(* IEC 61131-3 sources: Dev/Dev_V200/200 (part 15) *)

(* ---- _Nh_Frm_BRW.st ---- *)
FUNCTION _Nh_Frm_Row_BRW {HIDDEN}    : BOOL        // naplni, alebo refreshne objekty jedneho riadka browsu/frame/home
	{ $ IFDEF __NH_WEB }
   VAR_INPUT
      new   : BOOL;
      row   : USINT;
   END_VAR
   VAR_TEMP
		blk	: USINT;
      cp    : USINT;
//      np    : INT;
   END_VAR
   _Nh_Frm_Row_BRW := true;
   IF new THEN
		cp := xR^.h.cf.c;
      IF xL^.obj = 11 AND xR^.h.cf.c = 1 THEN                                           // ZONA domcek       1 ZON -> ROMs
			cp := 3;
		ELSIF xR^.h.new  THEN
			new := false;
      END_IF;
		IF new THEN
      	_Nh_Brw_Row_DSH(row := row, frm := USINT_TO_UINT(aCfg[ cp ].fBr) );   	// nacita FRM a podla DSH pripravi korekcie X,Y
			_Nh_Brw_Row_OBJ(row := row);
	      _Nh_FRM_Read(frm:=246);   	// nacita rozne preddefinovane objekty v riadku	 xR^.o.ob[]
	     	_Nh_Chk_FAV();
   	   CASE xR^.h.cf.c OF
			 0:	;
			50:	// timer - v priebehu refreshu sa nemeni
					xTim	:= xDev;
					memcpyPTR(length:=SIZEOF(NH_OBJ_DAT), source:=ADR(yFrm_246.tim_1), dest:=ADR(xR^.o.ob[6]) );		// nastavi zobrazovanie obrazka typu casovaca nad hlavnou ikonou
					memcpyPTR(length:=SIZEOF(NH_OBJ_DAT), source:=ADR(yFrm_246.e4O1), dest:=ADR(xR^.o.ob[7]) );		// vypne zobrazovanie na stavovou ikonou
			 		x4o   			:= ADR(xR^.o.ob[6]);
					x4o^.obr[2]    :=	yFrm_246.tim_1_typ_obr[ xTim^.cf.typ ];			// podla typu vyberie obrazok
					blk	:= 5;
	      END_CASE;

	   END_IF;
	END_IF;

   CASE xR^.h.cf.c OF

   	0: ;
    	1:	_Nh_Shw_ROM_ROW();
		2: // CAT
		   	_Nh_FRM_Read(frm:=232);
            xR^.o.ob[5].cf.c := 0;
  	         xR^.o.ob[5].cf.n := yFrm_232.cat[xR^.h.cf.n].txt;                                  // cislo textu v 1.riadku
            xR^.o.ob[6].cf.c := 0;
  	         xR^.o.ob[6].cf.n := yFrm_232.cat[xR^.h.cf.n].txt+1;                                  // cislo textu v 2.riadku je za prvym
				IF yFrm_232.cat[xR^.h.cf.n].cmd4 = 0 THEN
					xR^.o.ob[4].wh := 0;
				ELSE
					xR^.o.ob[4].cm := yFrm_232.cat[xR^.h.cf.n].cmd4;
				END_IF
				IF yFrm_232.cat[xR^.h.cf.n].cmd2 = 0 THEN
					xR^.o.ob[2].wh := 0;
				ELSE
					xR^.o.ob[2].cm := yFrm_232.cat[xR^.h.cf.n].cmd2;
				END_IF
				xR^.o.ob[1].cm := yFrm_232.cat[xR^.h.cf.n].cmd1;

            IF xA^.usr= 1 THEN                                                   // pre admina vypise cislo CAT
               xR^.o.ob[7].wh    := 6;
               xR^.o.ob[7].cf.c  := 254;
               xR^.o.ob[7].fmt   := CONCAT(INT_TO_STRINGF(xR^.h.cf.n,'%2u'), '');
            END_IF;
		3:	xR^.o.ob[9].cf.c:=252;										// vypisuje sa nazov domceka (domovskej zony)
				_Nh_Shw_ROM_ROW();
		6: // HET
  				xHet  	:= xDev;
				IF xL^.dsh = 4 THEN
					_Nh_Shw_CPY();
      		ELSE
					_NH_Het_Map_Reg();
//					IF xHet^.io[0].own THEN                // DEV regulovanej teploty
               	IF xRegMod^.wht = 1 THEN
							xR^.o.ob[2].fmt := REAL_TO_STRINGF(xHet^.al.ou.val,'%5.1f°');
						ELSE
							xR^.o.ob[2].fmt := REAL_TO_STRINGF(xHet^.al.ou.val,'%5.0f %%');
						END_IF
//					END_IF ;
					IF xHet^.io[1].own THEN                // ma termoventil
						IF xHet^.io[1].zon THEN             // TVE ma teplotu
							xR^.o.ob[5].fmt := REAL_TO_STRINGF(xHet^.io[1].val,'%5.1f°');
						ELSE
						   xR^.o.ob[5].wh := 0;
						END_IF;
						xHet^.al.lst := true;
					ELSE
		   			xR^.o.ob[5].wh := 0;
						xHet^.al.lst := false;
					END_IF;
//	 			IF xA^.admin = false THEN
	 				IF xM^.set=false OR xA^.UsrRight < 2 THEN
	 					xR^.o.ob[1].cm   := 0;
 						xR^.o.ob[4].fn   := 0;
 						xR^.o.ob[6].fn   := 0;
					END_IF;
				END_IF;
  		47: // HEV
            xHet  := xDev;
				IF xL^.dsh = 4 THEN
					_Nh_Shw_CPY();
         	END_IF;
      		IF xHet^.io[0].own THEN                // aktualne % CO2 zo snimaca
					xR^.o.ob[2].fmt := REAL_TO_STRINGF(xHet^.io[0].val,'%6.0f %%');
				END_IF;
				IF xHet^.io[2].own THEN                // ma termoventil
					xHet^.al.lst := true;
				ELSE
					xHet^.al.lst := false;
				END_IF;
//  	 			IF xA^.admin = false THEN
	 			IF xM^.set=false OR xA^.UsrRight < 2 THEN
 					xR^.o.ob[1].cm   := 0;
	 				xR^.o.ob[4].fn   := 0;											// setup nie je
 					xR^.o.ob[6].fn   := 0;                               	// lst vazby nie su
  				END_IF;
				IF xL^.chk AND xR^.o.ob[4].cf.c > 0 THEN
					IF acfg[xR^.o.ob[4].cf.c].tgrp = 15 THEN
 						xR^.o.ob[7].wh   := 0;                      			// ked je vo vazbe PIR, vypnu sa predvolby a zobrazuju sa prvky PIR
					END_IF;
				END_IF;

		7: // KOT
 			_Nh_Shw_TVE_ROW();

		8: // TVE
 			_Nh_Shw_TVE_ROW();

		9: // CER
 			_Nh_Shw_TVE_ROW();

		15: //PIR
				IF	xR^.h.pir THEN					// je vo vazbe
					;
				ELSIF	_NhxRom(nr := xDev^.cf.rom ,x:=55) THEN
					_Nh_Shw_107_ROM(o:=7, day:=true);
	            _Nh_Frm_STA_OU(obj:=2, o:=8);
					blk	:= 5;
//   				_Nh_DEF_VAR(wh:=20, o:=6, x:=ADR(xDev^.cf.blk) );
				ELSE
					xR^.o.ob[7].wh		:= 0;
				END_IF;

		23: // REK
				 _Nh_Shw_TVE_ROW();

		31: // ROL
				xRol 		:= xDev;
				IF new  THEN                        // pri prvom vstupe do FRM. nacitat iny formular podla menu. n
					xRo		:= ADR(xR^.o.ob[5]);
					IF xR^.h.cf.p=0 THEN
						xR^.h.cf.p := xRol^.cf.par;
					END_IF;
					xRo^.cf	:= xR^.h.cf;
					xRo^.chk	:= xL^.chk;					// priznak vazby
				END_IF;

  	 			IF xM^.set AND xF^.cf.c = 2 AND xF^.cf.n = 3 THEN		// pristupne kopirovanie
		  	 			IF xU^.o[1].fn  = 44 AND xL^.dsh = 1 THEN									// zlte COPY
//      D1_7       : NH_OBJ_4O1 	:= (obj:=1, obr:=[44,38,0,0], cmd:=[0,0,0,0], wxy:=[0,0,0,0],ok:=[0,0,0,0], txt:=[0,0,0,0],  );                          // 5=slider;
//							xR^.o.ob[7]		:= xR^.o.ob[8];
						 	x4o    			:= ADR(xR^.o.ob[8]);
							xR^.o.ob[1].cm 	:= 128;									// click na hlavnu ikonu = oznacovanie
							xR^.o.ob[10].cm 	:= 128;									// nazov
							x4o^.wh			:= 107;
							x4o^.obj			:= 1;
   	 					x4o^.wxy[1]    := 52;
    						x4o^.wxy[2]    := 42;
							x4o^.obr[1]		:= 44;
							x4o^.obr[2]		:= 38;
							x4o^.ok[1] 		:= xU^.o[1].wh = xR^.h.cf.n;
							x4o^.ok[2] 		:= xRol^.me.cpy;
						ELSE
							xR^.o.ob[1].cm 	:= 204;                         	// standardne parametre rolety
							xR^.o.ob[10].cm 	:= 204;								// nazov
							x4o^.wh				:= 0;
						END_IF;
				END_IF;

		131: // ROL
            xRol     := xDev;
				IF new THEN
	            ix       := xR^.o.ob[6].fn;                                             // slider je v 8
   	         xS       := ADR(xB^.s[ix]);
		         _NhSetObjBrw(ob:=5, wh:=24, w:=50,  t:=4, c:=1, cm:=48,  vb := ADR(xRol^.cx.SetLam),   fmt := '119500');        // ROL/LAM
         	   _Nh_Frm_Row_O13(ob:=6, vb:= PTR_TO_UDINT( ADR(xRol^.al.in.Val) ) );
	  	 			IF xM^.set AND xF^.cf.c = 2 AND xF^.cf.n = 3 THEN		// pristupne kopirovanie
		  	 			IF xU^.o[1].fn  = 44 THEN									// zlte COPY
//      D1_7       : NH_OBJ_4O1 	:= (obj:=1, obr:=[44,38,0,0], cmd:=[0,0,0,0], wxy:=[0,0,0,0],ok:=[0,0,0,0], txt:=[0,0,0,0],  );                          // 5=slider;
							xR^.o.ob[7]		:= xR^.o.ob[8];
						 	x4o    			:= ADR(xR^.o.ob[7]);
							xR^.o.ob[1].cm := 128;									// click na hlavnu ikonu = oznacovanie
							x4o^.wh			:= 107;
							x4o^.obj			:= 1;
   	 					x4o^.wxy[1]    := 52;
    						x4o^.wxy[2]    := 42;
							x4o^.obr[1]		:= 44;
							x4o^.obr[2]		:= 38;
							x4o^.ok[1] 		:= xU^.o[1].wh = xR^.h.cf.n;
							x4o^.ok[2] 		:= xRol^.me.cpy;
						ELSE
							xR^.o.ob[1].cm := 204;                         	// standardne parametre rolety
							x4o^.wh			:= 0;
						END_IF;
					END_IF;
				 	x4o    			:= ADR(xR^.o.ob[8]);
					x4o^.wh			:= 107;
					y4o := x4o^;
					IF xRol^.cx.yLam <= 0.0 THEN
						x4o^.obr[1]		:= 500;
					ELSIF xRol^.cx.yLam >= 100.0 THEN
						x4o^.obr[1]		:= 502;
					ELSE
						x4o^.obr[1]		:= 501;
					END_IF;
					IF xRol^.cx.CMD = 12 THEN
						x4o^.ok[2]		:= true;										// zobrazi blokovanie vetrom
					ELSE
						x4o^.ok[2]		:= false;
					END_IF;

//					x4o^.obr[1]		:= 10000+REAL_TO_INT(xRol^.cx.yBli);			// namiesto obr sa vypise text = poziacia rolety
//					x4o^.obr[3]		:= 10000+REAL_TO_INT(xRol^.cx.yLam);			//

				END_IF;
				IF xRol^.cx.SetLam = false THEN								// slider ROL
//    				xR^.o.ob[6].BgC := 9;                              // modra
    				xR^.o.ob[6].BgC := 3;                              // modra
					IF xRol^.cx.CMD > 200 THEN
						xRol^.al.in.Val := xRol^.cx.yrol;
					END_IF;
				ELSE
//					xR^.o.ob[6].BgC := 10;                                	// biela pre LAM
					xR^.o.ob[6].BgC := 27;                                	// biela pre LAM
					IF xRol^.cx.CMD > 200 THEN
						xRol^.al.in.Val := xRol^.cx.yLam;
					END_IF;
         	END_IF;

		37: // GATE
				xGat	:= xDev;
            xR^.o.ob[5].fn := _Nh_O12(xGat^.cx.btn,69,66);                   // slider - aktivovana SCN je oranzova, inak zlta
				IF  xGat^.cf.typ < 2 THEN											// garaz,brana
					_Nh_Frm_Row_O13(ob:=6, t:=0, vb:=PTR_TO_UDINT( ADR(xDev^.al.ou.val) ));
				ELSE
					xR^.o.ob[6].wh := 0;
				END_IF;
				_Nh_Frm_STA_OU(obj:=2, o:=8);

		{$IFDEF __NH_DALI}
		42: // DL-M
   	         xDlm              := xDev;
      	      ix                := xR^.h.cf.n;
         	   xDLfb             := ADR(aDali[ix]) ;
	            _Nh_Frm_Row_O13(ob:=5);

//    				xB^.s[ 0 ].v2 := 254.0;                         // ine ako DALI maju max 100%

   	         xPtD              := ADR(xR^.o.ob[9].cf.n);
      	      xPtD^             := PTR_TO_UDINT( ADR(xDlfb^.txt) );                   // v druhom riadku sa zobrazuje INFO o aktualnom parametre
         	   xR^.o.ob[9].cf.c  := 253;                                               // hodnota v pointri
(*
            xR^.o.ob[8].fmt   := INT_TO_STRING(xR^.h.cf.n);                         // cislo DLM l hlavnej ikone
            xR^.o.ob[8].BgC   := _Nh_U12(xDlm^.cx.sta.Present,8,1);                 // vykonany random/nevykonany
            xR^.o.ob[7].wh    := 0;
*)
	            xR^.o.ob[4].fn := _Nh_O12(xDlm^.cx.dlm.nShA>0,25,23 );                  // zeleny/sivy setup
//            xR^.o.ob[6].fn := _Nh_O12(xDLm^.al.lst,334,333);                  		// zeleny/sivy setup

      	      IF xDLm^.cx.sta.Err  THEN
         	      xDlfb^.txt := CONCAT(xDlfb^.txt,' E:');
            	   xDlfb^.txt := CONCAT(xDlfb^.txt,' '
               	                                                                     // RndAdr               Query
                  	                  ,USINT_TO_STRING(xDLm^.me.err.nErrS[1]),';'     // neprisla odpoved     Neprisla odpoved
                     	               ,USINT_TO_STRING(xDLm^.me.err.nErrS[2]),';'     // kolizia adries       Kolizia 2 adries
                        	            ,USINT_TO_STRING(xDLm^.me.err.nErrS[3]),';'     // niet co hladat
                           	         ,USINT_TO_STRING(xDLm^.me.err.nErrS[4]) );
	               xDlfb^.txt := CONCAT(xDlfb^.txt,'/'
   	                                 ,USINT_TO_STRING(xDLm^.me.err.nErrG[1]),';'
      	                              ,USINT_TO_STRING(xDLm^.me.err.nErrG[2]),';'
         	                           ,USINT_TO_STRING(xDLm^.me.err.nErrG[3]),';'
            	                        ,USINT_TO_STRING(xDLm^.me.err.nErrG[4]) );

//					ELSIF xDLfb^.cmd[1].cmd = 0 THEN
//	   	         xDlfb^.txt        := USINT_TO_STRINGF(xDlm^.cx.dlm.nSha,'%2d');         // pocet SHA
					ELSE
//	   	         xDlfb^.txt        := USINT_TO_STRINGF(xDlfb^.cmdQue,'%2u');         // pocet SHA
	            END_IF;
   	         // skupina
      	      // nazov DLM
         	   xR^.o.ob[10].cf   := xR^.h.cf;
	            x4o            := ADR(xR^.o.ob[7]);
   	         x4o^.obr[1]   := USINT_TO_INT( xDlm^.cx.dlm.nShA );
      	      IF xDLm^.cx.sta.Present = false THEN
         	      x4o^.BgC[1] := 2;
	            ELSE
   	            x4o^.BgC[1] := 3;
      	      END_IF;
		         x4o^.ok[2]        := 1;
      	      x4o^.obr[2]       := xR^.h.cf.n;

	            IF xDLm^.me.err.nErrS[2] > 0 THEN
   	            x4o^.ok [3] := 1;
      	         x4o^.obr[3] := USINT_TO_INT( xDLm^.me.err.nErrS[2] );
         	   ELSE
            	   x4o^.ok[3]        := 0;
	            END_IF;

      43: 	// DLS
    	      // xL^.obj :
				// 47 DLm/DLg
				// 48 DLm/DLs

				// 43 v hlavicke je toto 	DLs riadok je DLg 		priradzuje sa DLs->DLg
				// 44 v hlavicke je 			DLg riadok je toto DLs  priradzuje sa DLs->DLg
				xDLs     := xDev;
	         dlsl     := _Nh_DL_sha(nd := xR^.h.cf.n);
   	      dlma     := _Nh_DL_sha(ma := true, nd := xR^.h.cf.n);
				IF new THEN
	            x4o   := ADR(xR^.o.ob[7]);
					IF xM^.set AND xA^.UsrRight > 2 THEN
						x4o^.wh			:= 107;
	   	         x4o^.obr[1]   	:= USINT_TO_INT( dlsl );
  	      	      IF xDLs^.cx.sta.Present = false THEN
     	      	      x4o^.BgC[1] := 2;
      	         ELSE
  	      	         x4o^.BgC[1] := 5;
     	      	   END_IF;
        	      	IF xDLs^.cx.sta.ErrID > 0 THEN
           	      	x4o^.ok [3] := 1;
               	   x4o^.obr[3] := USINT_TO_INT( xDLs^.cx.sta.ErrID );;
	                  xR^.o.ob[0].FgC := 7;                                 				// cela dlazdica bude cevena
  		            ELSE
     		            x4o^.ok[3]        := 0;
        		         xR^.o.ob[0].FgC   := 1;
           		   END_IF;
	               x4o^.ok[2]  := 1;
  		            x4o^.obr[2] := USINT_TO_INT( dlma );

						IF xR^.h.chk  = false  THEN                                 		// len ked nie je vo vazbach
							xR^.o.ob[5].w  	:= 300;        											// skrati slider {mozno ho out5inOne aj tak prepise}
							xR^.o.ob[6] 		:= _NhBrwObj.dlgl;										// obrazok vseobecneho listu
							IF xDLs^.cx.scn.grp<>_eBtn15 THEN
  	   						xR^.o.ob[6].fn   	:= 334;
							ELSIF xDev^.al.lst THEN
     							xR^.o.ob[6].fn   	:= 192;
							ELSE
     							xR^.o.ob[6].fn   	:= 39;
							END_IF;
						END_IF;
					ELSE
						x4o^.wh			:= 0;
					END_IF;

						IF xDls^.cx.cfg.out5inOne THEN
							xR^.o.ob[5] 		:= _NhBrwObj.rgbwa;										// RGBWA namiesto slidera
							xR^.o.ob[5].wh		:= 121;
							xR^.o.ob[4].fn		:= 124;
							xR^.o.ob[4].cm		:= 74;	                                       // otvori priradenie RGBWA k DEV
							xR^.o.ob[2].cm 	:= 249;														// posle prikaz ON/OFF pre 5in1, hoci je aj chk
						END_IF;

					IF xR^.h.chk THEN
						_NhxPt(c := xF^.cf.c, n := xF^.cf.n,x:=432);
						IF xF^.cf.c = 44 THEN                                			// do DLg
							// DLs v scene nema parameter, nastavuje sa len LVL v strukture
	     					dlgr := _Nh_DL_sha(gr:=1,nd := xF^.cf.n)-100 ;				// 0..15
							_Nh_Frm_Row_O13(ob:=5, t:=1, vb:=PTR_TO_UDINT(ADR(xDLs^.cx.scn.LVL[ dlgr ])) );
							xR^.o.ob[2].cm 	:= 0;
						ELSIF xDls^.cx.cfg.out5inOne THEN
							IF xF^.cf.c = 8 THEN													// zatial len pre TVE
								xR^.o.ob[6] 		:= _NhBrwObj.srgbwa;							// led na sebe = ktory port {RGBWA} je priradeny k DEV v hlavicke
								xR^.o.ob[6].cm 	:= 251;											// posle prikaz ON/OFF pre 5in1
								_NhxPt(c:=xF^.cf.c, n:=xF^.cf.n, x:=-154);
								xTve := xPt;
								_Nh_DEF_VAR(wh:=20, o:=6, x:=ADR(xTve^.io[0].dev.o));
							ELSE
								xR^.o.ob[6].wh 	:= 0;											// nebude zobrazovat vyber konkretnej farby
							END_IF;
						ELSIF _Nh_IO_MAP(cIo:=xF^.cf.c, Dev:=xR^.h.cf.c)  THEN
							_Nh_Frm_Row_O13(ob:=5, t:=0, vb:=PTR_TO_UDINT(ADR( xPtIOa^.val ) ));
							xR^.o.ob[2].cm 	:= 0;
						ELSIF xR^.o.ob[4].cf.c = 15 THEN                                				// check PIR ma prednost
      					xR^.o.ob[5].wh 	:= 0;
						ELSIF _NhxPar(cp := aCfg[xR^.h.cf.c].par , np := xR^.h.cf.p,x:=-1006) THEN		// SCN,ACT,BLK
							_Nh_Frm_Row_O13(ob:=5, t:=1, vb:=PTR_TO_UDINT(ADR(xPar^.all.lvl)) );
						ELSE
							xR^.o.ob[5].wh := 0;
							xR^.o.ob[2].cm := 0;
						END_IF;

(*
					ELSIF xDls^.cx.cfg.out5inOne THEN								// do TVE, bude zobrazena RGBWA +
						xR^.o.ob[5] 		:= _NhBrwObj.rgbwa;											// obrazok vseobecneho listu
						xR^.o.ob[5].wh		:= 121;
						xR^.o.ob[2].cm 	:= 249;													// posle prikaz ON/OFF pre 5in1
*)
					END_IF;

				ELSIF	xR^.h.chk THEN
						IF xF^.cf.c = 44 THEN                                		// do DLg
      					dlgr := _Nh_DL_sha(gr:=1,nd := xF^.cf.n)-100 ;				// 0..15
							IF  xR^.o.ob[2].tch THEN												// prepnut LVL s status - LVL je uz zapisany v parametri
								xDLs^.cx.scn.LVL[ dlgr ] := xPar^.all.lvl;
							END_IF;
							IF xR^.o.ob[2].tch OR (xR^.o.ob[5].tch AND xA^.tch.Qf) THEN
//		                  _Nh_DL_ADD_Task(wht:=  4, par:= 1, sha := dlsl , val := dlGr+100, dlm := dlma  );	// prida ballast do sceny, hoci tam uz moze byt
//      		            _Nh_DL_ADD_Task(wht:=102, par := dlgr,  	//   scena		0..15                    	// nastavi LVL pre ballast v scene
      		            _Nh_DL_ADD_Task(wht:=2, par := dlgr,  	//   scena		0..15                    	// nastavi LVL pre ballast v scene
         	                                   	sha := dlsl,    //   ballast	0..63
            	                                	val := REAL_TO_USINT(USINT_TO_REAL(xDLs^.cx.scn.LVL[ dlgr ])*2.45) ,
               	                             	dlm := dlma );
							END_IF;
						END_IF;
				ELSIF xDls^.cx.cfg.out5inOne THEN								// do TVE, bude zobrazena RGBWA +
					;
//					xR^.o.ob[4].fn	:= 124;
//					xR^.o.ob[4].cm	:= 76;

				ELSE
					_Nh_Frm_Row_O13(ob:=5, t:=0, vb:=PTR_TO_UDINT(ADR(xDev^.al.in.val)) );
				END_IF;

				IF xDls^.cx.cfg.out5inOne THEN
						;
				ELSE
					_Nh_Frm_STA_OU(obj:=2, o:=8);											// ikony nad stavovym obrazkom
				END_IF;

      44: // DLg
			      // 56:  DLs ->  DLg		... v hlavicke je DLsa v riadkoc su sceny do ktorych moze ist
				   xDLg     := xDev;
   	         dlma     := _Nh_DL_sha(gr:=1, ma := true, nd := xR^.h.cf.n);            // master
      	      dlgr     := _Nh_DL_sha(gr:=1, nd := xR^.h.cf.n)-100;                    // cislo GRP - 100 prevedie na 0..15
					xDLg^.al.lst	:= xDLg^.cx.Sta.Present;											// dolezitejsi je Present, je aj po restarte aktivny
	            x4o   := ADR(xR^.o.ob[7]);
       			IF xR^.h.chk  THEN
						IF xF^.cf.c = 43  THEN																// DLs v hlavicke do tejto sceny
							IF _NhXPt(c:=xF^.cf.c, n:=xF^.cf.n,x:=-135) THEN
								xDLs := xPt;
					         dlsl     := _Nh_DL_sha(nd := xF^.cf.n);
								_Nh_Frm_Row_O13(ob:=5, t:=1, vb:=PTR_TO_UDINT(ADR(xDLs^.cx.scn.lvl[dlgr])) );
								IF (xR^.o.ob[5].tch AND xA^.tch.Qf) THEN
      			            _Nh_DL_ADD_Task(wht:=2,par := dlgr,  	//   scena		0..15                    	// nastavi LVL pre ballast v scene
         		                                   sha := dlsl,    //   ballast	0..63
            		                                val := REAL_TO_USINT(USINT_TO_REAL( xDLs^.cx.scn.LVL[ dlgr ])*2.45),
               		                             dlm := dlma );
								END_IF;
							ELSE
								xR^.o.ob[5].wh := 0;
							END_IF;
						ELSIF xR^.o.ob[4].cf.c <>  15 THEN
		         	   _Nh_Frm_Row_O13(off:=xR^.h.pir, ob:=5);
						END_IF;

					ELSE
	         	   _Nh_Frm_Row_O13(off:=xR^.h.pir, ob:=5);
//		            xR^.o.ob[5].BgC := _Nh_U12(xDLg^.al.ou.val=254.0,6,5);                   // slider - aktivovana SCN je oranzova, inak zlta
		            xR^.o.ob[5].BgC := _Nh_U12(xDLg^.al.ou.val=100.0,6,5);                   // slider - aktivovana SCN je oranzova, inak zlta
					END_IF;

					IF xM^.set AND xA^.UsrRight > 2 THEN
							x4o^.wh	:= 107;
      		         x4o^.obr[1]   := USINT_TO_INT( dlgr );
         		      IF xDLg^.cx.sta.Present = false THEN
            		      x4o^.BgC[1] := 2;
	          	     	ELSE
   	         	      x4o^.BgC[1] := 6;
	   	            END_IF;
   	   	         IF xDLg^.cx.sta.ErrID > 0 THEN
      	   	         x4o^.ok [3] := 1;
         	   	      x4o^.obr[3] := USINT_TO_INT( xDLg^.cx.sta.ErrID );;
            	   	   xR^.o.ob[0].FgC := 7;                                 // cela dlazdica bude cevena
	               	ELSE
		                  x4o^.ok[3]        := 0;
   		               xR^.o.ob[0].FgC   := 1;
      		         END_IF;
         		      x4o^.ok[2]  := 1;
            		   x4o^.obr[2] := USINT_TO_INT( dlma );

                  IF xR^.o.ob[4].cf.c = 15 THEN
   			         xR^.o.ob[5].wh 	:= 0;
						ELSIF xR^.o.ob[6].wh <> 1 THEN
   						xR^.o.ob[6] 		:= _NhBrwObj.list;											// obrazok vseobecneho listu
	     	            xR^.o.ob[6].fn   	:= _Nh_O12(in := xDev^.al.lst , o1:=192, o2:=39); // LIST zeleny/sivy
						   xR^.o.ob[5].w  	:= 300;        												// skrati slider
						END_IF;

   				ELSE
						x4o^.wh	:= 0;
   				END_IF;

(*
					IF NOT( xR^.o.ob[4].cf.c = 15 AND xR^.h.chk ) THEN
						xR^.o.ob[6].wh	:= 1;															// ked je vo vazbe PIR
   				END_IF;
*)
      	      IF xDlg^.cf.rom = 0 THEN
         	      xR^.o.ob[9].wh := 0;
	            END_IF;
            	// 53 DLs/DLg
					_Nh_Frm_STA_OU(obj:=2, o:=8);

		{$ELSE}
	        	42: // DL-M
					;
  				43: // DLS
					;
	        	44: // DL-M
					;
		{$END_IF}

	  48:	// ALA
   		xAla  := xDev;
   		_NhxZon(nz:=xAla^.cf.rom);
	   	xR^.o.ob[4].cm := 204;
   		IF xZon^.cx.lck.stat = SINT_TO_USINT(xAla^.cf.typ) THEN
		   	xR^.o.ob[0].FgC := 3;
    			xR^.o.ob[0].BgC := 1;
			END_IF;

	 150: //TIMER
			xTim	:= xDev;
//			xR^.o.ob[6] 		:= _NhBrwObj.rgbwa;	//_NhBrwObj.dlgl;										// obrazok vseobecneho listu
//_NhBrwObj.dlgl
//			xR^.o.ob[7] 		:= _NhBrwObj.tim_1;										// obrazok vseobecneho listu
	 		x4o    			:= ADR(xR^.o.ob[7]);
			IF xTim^.cf.typ < 2 THEN

(*

						 	x4o    			:= ADR(xR^.o.ob[7]);
							xR^.o.ob[1].cm := 128;									// click na hlavnu ikonu = oznacovanie
							x4o^.wh			:= 107;
							x4o^.obj			:= 1;
   	 					x4o^.wxy[1]    := 52;
    						x4o^.wxy[2]    := 42;
							x4o^.obr[1]		:= 44;
							x4o^.obr[2]		:= 38;
							x4o^.ok[1] 		:= xU^.o[1].wh = xR^.h.cf.n;
							x4o^.ok[2] 		:= xRol^.me.cpy;

				_Nh_Shw_107_ROM(off:=1, o:=7);			// vypne zobrazenie nad hl.obrazkom
*)       END_IF;
				_Nh_Shw_107_ROM(off:=1, o:=8);
				blk	:= 5;

      ELSE
         IF xR^.h.cf.c > 0 THEN
				IF aCfg[xR^.h.cf.c].fbr = 15 THEN											// PODLA FORMULARA BROWSU
              	// DOR
						blk	:= 5;
						IF xA^.admin  THEN
						ELSE
                     xR^.o.ob[6].wh :=  0;                        // u WSB vypne predvolby
                     xR^.o.ob[2].cm :=  0;                        // u WSB vypne predvolby
						END_IF;
              ELSIF aCfg[xR^.h.cf.c].fbr = 20 THEN
					  // LUX,TER,TEH,TEK, 41=CO2
						_Nh_Shw_B20_ROW();
   					blk	:= 6;
	           ELSIF 	aCfg[xR^.h.cf.c].fbr = 43 							// SVD,SVA,RGB,ZAS,32=SIR,49=VVO
	           		OR aCfg[xR^.h.cf.c].fbr =  5 THEN					// SCN,ACT,DLS,DLG,DLM
		            _Nh_Frm_STA_OU(obj:=2, o:=8);
						IF aCfg[xR^.h.cf.c].analog THEN
		         	   _Nh_Frm_Row_O13(off:=xR^.h.pir ,ob:=5);
						ELSIF xM^.set THEN
//							blk 					:= 5;
							xR^.o.ob[5].wh    := 0;
						ELSE
							xR^.o.ob[5].wh    := 0;
						END_IF;
            ELSE
            ;
            END_IF;
      	END_IF;
	END_CASE;

	IF xM^.set AND new AND blk > 0 THEN
		_Nh_DEF_VAR(wh:=20, o:=blk, x:=ADR(xDev^.cf.blk));

//		xR^.o.ob[blk].x     := 125;
		xR^.o.ob[blk].w     := 48;
		xR^.o.ob[blk].h     := 48;
		xR^.o.ob[blk].FgC   := 4;
		xR^.o.ob[blk].BgC   := 2;
		xR^.o.ob[blk].fn    := 0;

	END_IF;

	{$ END_IF }
END_FUNCTION

(* ---- _Nh_Frm_HOM.st ---- *)
{ $ IFDEF __NH_WEB }

FUNCTION _Nh_Map_Idx  {HIDDEN}  : BOOL     // premapuje xIdx (Veta browsu (ixb) v wrk pamati ) podla zvolenej sady indexu (ixb), pripadne vycisti browser
   VAR_INPUT
      ini   : BOOL;                       // vymaze data browsu aj indexov
      ixb   : USINT:= 0;                  // sada dat
      idx   : USINT:= 1;                  // cislo vety (index v sade dat), ktoru ma namapovat (0=1.veta)
   END_VAR
   xIxB  := ADR(xM^.ixb[ixb]);
   IF ini THEN
      IF ixb > 0 THEN
         xIxB^.ofs := xM^.ixb[ixb-1].ofs + xM^.ixb[ixb-1].idx;
//         xIxB^.row.rws   := 6;                                                // len pre Quick menu
      ELSE
         _NheBrw( wht := 4);                                                  // vymaze kompletny browser aj s IX
         xIxB^.row   :=_NhDsh.dsh[xL^.dsh];                                   // nastavi riadky aj
      END_IF;
   END_IF;
   sz          := SIZEOF(NH_IDX) * USINT_TO_UDINT( xIxB^.ofs + idx - 1 ) ;
   xIdx        := ADR(mRam[aSys.vIx1]) + sz;    // za poslednu vetu zo vsetkych vazieb
   _Nh_Map_Idx := xIxB^.idx > 0;

END_FUNCTION

//FUNCTION _NhFinIdx {HIDDEN} : USINT    // najde v indexe DEV ulozene v 1.riadku, alebo prida a uberie zadany pocet riadkov s nastavi tak 1.riadok

FUNCTION _Nh_Chk_RoW   {HIDDEN}  : BOOL    //
   VAR_INPUT
      chk   : BOOL;                                   // posun dohora (dalej ) o pocet riadkov row
      vaz   : BOOL;
   END_VAR
   _Nh_Chk_RoW := false;
   IF xL^.fvz THEN
      xM^.wht := 20;                                           // nove data, vypis od zaciatku
      RETURN;
   END_IF;
   i := 0;                                   //
   xM^.wht := 25;                                              // novy index, vypis od zpamatanej vety v 1.riadku
   IF chk THEN                                                 // zaskrtnutie
      IF vaz AND xL^.fdv = 0 THEN                              // veta je VAZ[2] a nie je zapnuty filter na DEV = nevieme kde v browse sme
         xL^.rw1 := xR^.h.cf;                                  // check veta sa nastvi na 1.riadok
      END_IF;
   ELSIF vaz THEN
      IF xA^.tch.row = 1 THEN
         IF xIxB^.ix2 > xIxB^.ix1 THEN
            i := xIxB^.ix1 + 1;
         ELSIF xIxB^.ix1 > 1 THEN
            i := xIxB^.ix1 - 1;
         ELSE
            xM^.wht := 20;
         END_IF;
      END_IF;
//   ELSE
//      xM^.wht := 10;
   END_IF;
   IF i > 0 THEN
      _Nh_Map_Idx(idx:=i);
      xL^.rw1     := xIdx^.ix[aWeb.nbr].dev;       // check vazby presunie na 1.riadok                            //
   END_IF;
END_FUNCTION

FUNCTION _NhSet1Row {HIDDEN}  : BOOL    // najde v indexe DEV ulozene v 1.riadku, alebo prida a uberie zadany pocet riadkov s nastavi tak 1.riadok
   VAR_INPUT
      up    : BOOL;                                   // posun dohora (dalej ) o pocet riadkov row
      dn    : BOOL;                                   // posun dolu   (spat) o pocet riadkov row
      end   : BOOL;                                   // pokusi sa zaradit pridavanu vetu n koniec browsu
      del   : BOOL;                                   // zisti, ci nedoslo k vymazaniu vety v 1.riadku, ak ano prestavi na dalsiu alebo na prvy index
      fnd   : BOOL := true;                           // vzdy sa hlada
      ixb   : USINT := 0;                             // indexova sada 0,1
      row   : USINT;                                  // prida, alebo uberie riadky, ak sa najde pozadovana veta
   END_VAR
   _NhSet1Row := false;
   rb := _Nh_Map_Idx(ixb := ixb);                                               // namapuje 1.index
   xIxB^.ix2   := 0;                                                    // tu sa vkladaju data do ROW
   IF fnd THEN
      FOR i := 1 TO xIxB^.idx DO                                        // prechadza vsetky indexy
         IF xL^.rw1.c  = xIdx^.ix[aWeb.nbr].dev.c AND
            xL^.rw1.n  = xIdx^.ix[aWeb.nbr].dev.n THEN
            _NhSet1Row := true;
            IF end THEN
               IF i <= xIxB^.row.rws THEN
                  i := 1;
               ELSE
                  i := i - xIxB^.row.rws + 1;
               END_IF;
            END_IF;
            EXIT;
         END_IF;
         xIdx  := xIdx + SIZEOF(NH_IDX);
      END_FOR;
   ELSIF xIxB^.ix1 > 0 THEN                                             // nehlada sa. nastavi prva veta zobrazena v browse
      i           := xIxB^.ix1;
      _NhSet1Row  := true;
   ELSE
      i  := 1;
   END_IF;
   IF xIxB^.idx = 0 THEN
      xIxB^.ix1 := 0;                                                   // nemame data
      RETURN;
   ELSIF xIxB^.idx <= xIxB^.row.rws THEN                                // mame menej dat ako jedna stranka riadkov
      i   := 1;
   ELSIF _NhSet1Row THEN
      IF del THEN                                                       // v indexe sa nasla veta z 1.riadku
         IF _NhxDev(c := xL^.rw1.c, n := xL^.rw1.n, x:=10) = false THEN      // veta v 1.radku bola prave vymazana
            IF xIxB^.idx <= i THEN                                      // tato veta je posledna
               i := 1;                                                  // bude sa vypisobvat kompletny vypis
            ELSE
               i := i + 1;                                              // nastavi sa nasledujuca veta
            END_IF;
         END_IF;
      ELSIF dn THEN
         i := MAX(1,i - MIN( i, row )) ;                                // +1 aby sa nastavil riadok 1, nie 0;
      ELSIF up THEN
         i := i + row;                                                  // toto by mohol byt prvy riadok (za poslednym doterajsim)
         IF i + xIxB^.row.rws > xIxB^.idx THEN                          // ci po pridani riadkov, bude zaplnena cela stranka
            i := xIxB^.idx - xIxB^.row.rws + 1;
         END_IF;
      END_IF;
   ELSIF xIxB^.idx > 0 THEN                                             // nenasla sa veta, mame data, ide sa od zaciatku, nastavi sa 1.veta,
      i  := 1;
   END_IF;
   _Nh_Map_Idx(ixb := ixb, idx := i);                                     // namapuje najdeny index
   xIxB^.ix1   := i;                                                    //

   xL^.rw1     := xIdx^.ix[aWeb.nbr].dev;                                   //

   _NhSet1Row  := true;                                                 //

(*
   IF xIxB^.ix1 > 0 AND xIxB^.row.rws > 0 THEN
      xIxB^.n  := xIxB^.idx / xIxB^.row.rws;
      IF mod(xIxB^.idx,xIxB^.row.rws) > 0 THEN
         xIxB^.n  := xIxB^.n + 1;
      END_IF;
      IF xIxB^.n > 1 THEN                                                              // bude vykreslovat gulicky stran
         xIxB^.w  := 40;
         xIxB^.x1 := (x2 - USINT_TO_INT(xIxB^.n-1) * 40)/2;
      ELSIF xIxB^.n > 0 THEN                                                              // bude vykreslovat gulicky stran
         xIxB^.x1 := x2/2;
      END_IF;
//     xIxB^.pg  := 1;
   END_IF;
*)

END_FUNCTION

FUNCTION _NhVazErr {HIDDEN} : BOOL                // prida vetu do indexu browsu
   yTx2 := CONCAT(yTx2,' in: ',USINT_TO_STRINGF(xVaz^.in.c,'%3d'),';',INT_TO_STRINGF(xVaz^.in.n,'%4d'),';',INT_TO_STRINGF(xVaz^.in.p,'%3d'),';',
                       ' ou: ',USINT_TO_STRINGF(xVaz^.ou.c,'%3d'),';',INT_TO_STRINGF(xVaz^.ou.n,'%4d'),';',INT_TO_STRINGF(xVaz^.ou.p,'%3d') );
   rb := _Nh1RowTxt(logRst := 1,adTime := 3, EmpRow:=1);
END_FUNCTION

(*
FUNCTION _NhSbjOk {HIDDEN} : BOOL                // prida vetu do indexu browsu
   VAR_INPUT
      cf    : USINT;
      rom   : USINT;
   END_VAR
   _NhSbjOk := true;
   IF xA^.admin OR xA^.sbj = 1 OR rom = 0 THEN
      ;
   ELSIF cf = 1 THEN
      _NhSbjOk := rom = xA^.sbj OR rom = 4;
   ELSIF cf = 3 THEN
      _NhSbjOk := rom = xA^.sbj;  //  OR rom = 4;
   ELSIF _NhxPt(cf:=1, nd := USINT_TO_INT(rom), x:=85) AND xPt^.cf.rom > 0 THEN
      _NhSbjOk := xPt^.cf.rom = xA^.sbj ;
   END_IF;
END_FUNCTION
*)

FUNCTION _Nh_DEV_AL_VAZ {HIDDEN} : BOOL
	VAR_INPUT
		clr	: BOOL;
		i1		: USINT := 100;
		i2		: USINT := 100;
//		io		: PTR_TO NH_VAL_IO;
	END_VAR
	_Nh_DEV_AL_VAZ	:= true;
	IF clr THEN
		IF aCfg[cf].al > 0 THEN                                     // al ma /al, resetne priznak, IOX ho vrati

   		CASE cf OF
     			42 : ;
     			43 : ;
     			44 : ;
     		ELSE  xDev^.al.lst  := false;                            // lst sa vymaze len pre NE-DALI
     		END_CASE;
		END_IF;
	ELSE
		WHILE i1 <= i2 DO
			IF xPtIO^.dev.c > 0 THEN
				IF _NhxPt(c:=xPtIO^.dev.c, n := xPtIO^.dev.n,x:=-124) THEN
					;
				ELSE
					xPtIO^.dev.c 	:= 0;
				END_IF;
			END_IF;
			xPtIO := xPtIO + SIZEOF(NH_VAL_IO);
			i1 	:= i1+1;
   	END_WHILE;
	END_IF;
END_FUNCTION

(*
FUNCTION _NhSbjOk {HIDDEN} : BOOL                // prida vetu do indexu browsu
   VAR_INPUT
      cf    : USINT;
      rom   : USINT;
   END_VAR
   _NhSbjOk := true;
   IF xA^.admin OR xA^.sbj = 1 OR rom = 0 THEN
      ;
   ELSIF xL^.obj=0 THEN                                                 // HOME DASH
      ;
   ELSIF xL^.obj=2 THEN                                                 // FAV
     _NhSbjOk := rom = xA^.sbj;
   ELSIF xF^.cf.c=1 AND xF^.cf.n=0 THEN                                 // zoznam miestnosti
     _NhSbjOk := rom = xA^.sbj;
   ELSIF xF^.cf.c=1 THEN                                                // 1.miestnost
      _NhSbjOk := true;
   ELSIF xF^.cf.c=3 OR (xF^.cf.c=2 AND xF^.cf.n=6) THEN                 // ZONE alebo SEC
      _NhSbjOk := rom = xA^.sbj OR rom = 4;
   ELSIF _NhxPt(cf:=1, nd := USINT_TO_INT(rom), x:=85) AND xPt^.cf.rom > 0 THEN
      _NhSbjOk := xPt^.cf.rom = xA^.sbj ;
   END_IF;
END_FUNCTION
*)

FUNCTION _Nh_Brw_Idx  {HIDDEN}  : BOOL                      (* VYTVORI ZOZNAM VIET PRE BROWSER VYHOVUJUCICH FILTRU *)
   VAR_INPUT
      ixb   : USINT  := 0;
   END_VAR
   VAR_TEMP
      io    : BOOL;
      dev   : BOOL;
      ix    : USINT;          // lokalne ix, nie globalne
      nx    : INT;
      xIdx1 : PTR_TO NH_IDX;
   END_VAR

   _Nh_Map_Idx(ini := true, ixb := ixb);
   xIdx1 := xIdx;                                              // zapamata si 1.vetu indexu
   _Nh_FRM_Read(frm:=235);                // typy DEV, Dev->Cat, Cat->Cat

      ix    := 1;
      cf    := _Nh_IxC[ix];                                    // vybrata veta CFG
      IF xL^.obj = 44 THEN                                     // BRW-DLg v hlavicke je 1.dali scena
         _NhxPt(c := xF^.cf.c, n := xF^.cf.n,x:=44);
         xDev2 := xPt;                                            // namapuje hlavicku do xDev2
      END_IF;

   IF xL^.vaz = 1 THEN                                         // FAV, xL^.fvz je vzdy true
      nd := 1;                                                                   //
      WHILE  nd  <= aVaz[xL^.vaz].Rec DO                                         // vsetky vety CFG
         IF _NhxVaz(cv := xL^.vaz, nd := nd ) THEN
            // oblubene
            // xA^.fav.c  ... user
            // xA^.fav.n = -1 dash menu
            // xA^.fav.n = -2 Quick menu
            // xA^.fav.n =  0 oblubene vsetkych usrov   (vtedy aj c:=0)
            // xA^.fav.n =  4 Quick setup
            // xA^.fav.n  > 4 konkretna veta v aCfg[20] ... oblubene pre usra c:=...
            // xVaz^.in.c ... podla xA^.fav.c ... user 0=vsetci
            // xVaz^.in.n ... podla xA^.fav.n
            IF xVaz^.in = xA^.fav THEN                         // zoznam FVL k vybratemu FAV v
               yIdxR      := _e_NH_IDX_ROW;
               yIdxR.fav  := true;
               yIdxR.dev  := xVaz^.ou;
               yIdxR.nd   := nd;
               yes        := true;
					cf 		  := xVaz^.ou.c;

					IF _NhxPtIO(c := xVaz^.ou.c, n := xVaz^.ou.n, x:=54) THEN
						xDev := xPt;
						_Nh_DEV_AL_VAZ(i1:=100, i2:=100 );
					END_IF;

            ELSE
               yes        := false;
            END_IF;
	         _NhCrIx(ok := yes);
         END_IF;
         nd := nd + 1;
      END_WHILE;
      cf    := 0;                                              // dalse sa nejde

   ELSIF xL^.obj=70 OR xL^.obj=71 THEN
		;
   ELSIF xL^.fvz AND xL^.vaz > 1 THEN
      cf    := 0;                                              // dalse sa nejde
   ELSE

   END_IF;

(*
   IF cf > 0 AND xF^.cf.c = 2 THEN                     // vstup do hlavnej urovne CAT
   	memset(val := 0, length := SIZEOF(NH_WRK_CAT), dest := VOID( aWeb.A[ aWeb.nbr ].cat ));        // vynuluje zoznam CAT pritomnych pre aktualny subj
		xF^.dev.n[ 0 ] := true;
   END_IF;
*)

   WHILE  cf > 0  DO        															// prechadza sa podla  _Nh_ixc[]. CAT [2] tam nie je
      IF xF^.dev.n[ cf ] OR xF^.dev.n[ 0 ] OR xF^.cf.c = 2 THEN   		// cf je v DEV liste alebo v hlavicke je CAT (DEV do browsu CAT)
         nx := 1;
      ELSE
         nx := 5000;
         cf := _Nh_CFG;                                                 // LEN poistka = nastavi sa na poslednu vetu CFG, ktura nema vety                 // vybrate CFG
      END_IF;

      WHILE nx <= aCfg[cf].Rec DO                                       // jedno CFG

			ok := xL^.obj=47 AND xU^.o[8].fn = 56;
         IF _NhxPt(c := cf, n := nx,x:=37) OR ok THEN
				xPtY	:= xPt;

(*//????12.12.23 nevieme na co ?
				IF _NhxPtIO(c := xVaz^.ou.c, n := xVaz^.ou.n, x:=55) THEN
					xDev := xPt;
					_Nh_DEV_AL_VAZ(i1:=100, i2:=100 );
				END_IF;
*)

				xDev := xPtY;
            sbj            := true;
            IF xF^.cf.c > 0 AND xF^.cf.n > 0 AND xF^.cf.c <> 2 THEN
               _NhxPt(c := xF^.cf.c, n := xF^.cf.n,x:=60);
               xDev2 := xPt;                                            // hlavicka
            ELSE                                                        // 0-ta uroven (FAV,ROM,CAT,ACT,SCN,SMW.....)
               xDev2 := xDev;                                           // toto je nespravne, len aby pointer neukazova do bludu (ked je v hlavicke
            END_IF;

            IF xDev^.ok.adm THEN                                        // len admin
               yes   := xA^.admin;
            ELSIF xDev^.ok.stp THEN                                     // len v rezime setup
               yes   := xM^.set;
            ELSE
               yes   := true;                                           // neobmedzeny pristup
            END_IF;
//				rom            := xF^.rom > 0 OR xF^.cf.c = 1 OR xF^.cf.c = 3;
				rom				:= true;
            nd             := nx;
            ok             := true;
            yIdxR          := _e_NH_IDX_ROW;
            yIdxR.dev.c    := cf;
            yIdxR.dev.n    := nd;
            yIdxR.dev.p    := xDev^.cf.par;

				IF xL^.vaz > 1 THEN
					xDev2^.al.vaz  := 0;
			   	xDev2^.al.lst  := 0;
				END_IF;

				IF xF^.cf.c = 2 THEN                                   			// browser CAT v hlavicke - prechadza DEV ine ako 2, ci sa zobrazia v CAT
	  				ok    := false;
					yes	:= yFrm_235.DevToCat[cf].n[xF^.cf.n];						// DEV sa zobrazuje aj v kategorii
					IF yes THEN
						IF xA^.CatOk = false THEN
							xA^.cat.cat[xF^.cf.n] := true;                        // oznaci CAT
						ELSIF xA^.cat.cat[xF^.cf.n] = false THEN
							yes := false;
						END_IF;
					END_IF;
	            _Nh_Chk_DALI();															// odfiltruje len dali do kategorie
				ELSIF cf = 2 THEN                                   				// CAT - v riadku
					yes := yes AND xF^.cat.n[cf];											// zaradi aj CAT
				ELSIF xDev^.cf.Idx <= 0 OR xDev^.cf.Idx > aCfg[cf].rec THEN    // nie je definovany index, alebo kekorektne data,  zostava cislo vety
               xDev^.cf.Idx := nd;
            ELSIF nx <> xDev^.cf.Idx THEN
               nd          := xDev^.cf.Idx;                                      // index je ukazuje na inu vetu. nx zostane, nd bude veta kam ukazuje index
               yIdxR.dev.n := nd;                                                // defaul sa pozije cislo vety
               ok          := _NhxPt(c := cf, n := nd,x:=38);
               xDev        := xPt;
            END_IF;

				IF xL^.obj=1 THEN                                           // FAV - zoznam oblubenych
                  xFav  := xDev;
                  //                                DSH,QCK,FV
                  yes   := Yes AND  (xA^.Admin OR
                                     xFav^.cx.n <= 0 OR
                                     xFav^.cx.c = xA^.usr);   // 0=vsetkych alebo konkretny FAV k usrovi
//                                     xFav^.cx.c = xA^.fav.c);   // 0=vsetkych alebo konkretny FAV k usrovi
				END_IF;

				IF ok THEN
               // kontrola konzistencie pre ROM,ZON
               CASE cf OF
                 1 : // ROM
							_Nh_TST_ROM();
                 3 : // ZON
							_Nh_TST_ZON();
							rom := false;
                 5 : // ACT
							IF xDev^.cf.rom > INT_TO_USINT(aCfg[3].Rec) THEN
	                     xDev^.cf.rom := 1;                  // naplni sa Rom = cislo vety
							END_IF;
               END_CASE;

	            IF _Nh_Chk_DALI() THEN ;
//						rom := false;
//	            ELSIF _Nh_Chk_SCN() THEN
					END_IF;

               IF xL^.chk THEN                                          // bude CHK, nie FAV
                  If yes THEN
                     IF _Nh_Chk_IODev() THEN
								rom := false;
							END_IF;
                     IF xL^.fvz THEN                                    // dev len s vazbou
                        yes := yes AND yIdxR.chk;
								rom := false;
                     END_IF;
                  END_IF;
               END_IF;

				END_IF;
				IF cf=1 OR cf=3 THEN
					xRom := xDev;

					xPtIO := ADR(xRom^.io[100]);
					_Nh_DEV_AL_VAZ(i1:=100,i2:=103 );														// oznaci al.vaz u DEV, ktore do ROM/ZON vstupuje DEV-vaz
				END_IF;

            // vo vacsine ROM podla hlavicky
            IF yes AND rom THEN
					IF  _Nh_Chk_IODev() THEN																		// otestuje ROM
						;
					ELSE
						;
					END_IF;
(*
					IF xF^.cf.c = 1 AND xF^.cf.n = USINT_TO_INT(_NhDefRom) THEN   			// default room
						yes := xDev^.cf.rom = _NhDefRom;
					ELSIF xF^.cf.c = 3 THEN																// 1. zona
						yes := xDev^.cf.rom = xF^.rom OR xL^.fvz = false;                 // riadok ma ten isty rom ako hlavicka
					ELSIF xL^.obj = 5  THEN   															// miestnosti
               	yes := true;
					ELSIF xF^.cf.c = 6 THEN
						yes := xF^.rom = 0 OR xDev^.cf.rom = xF^.rom;                         // riadok ma ten isty rom ako hlavicka
					ELSIF aCfg[cf].RomIsZone = false THEN
						yes := xF^.rom = 0 OR xDev^.cf.rom = xF^.rom;                         // riadok ma ten isty rom ako hlavicka
					ELSE
//						Yes := false;
					END_IF;
*)
            END_IF;
            // ak je uz DEV v indexe pridane z vazieb, uz sa nepridava
            If sbj THEN
//               yes := yes AND _NhSbjOK(cf:=yIdxR.dev.c ,rom := xDev^.cf.rom);;
            END_IF;
            // ON/OFF filter
            _Nh_Chk_OFF();
            _NhCrIx(ok := yes);
         END_IF;
         nx := nx + 1;
      END_WHILE;
      ix    := ix + 1;                                                           // presunie sa na dalsie CFG
      cf    := _Nh_IxC[ix];                                                     // vybrate CFG
   END_WHILE;

	// prechadza kategorie

//	xA^.CatOk := true;

   IF xF^.cf.c = 2 THEN                                              			// do CAT v hlavicke prida aj podkategorie
		xA^.cat.cat[35] := true;																// dali
		IF xA^.CatOk = false THEN
			FOR cf := 1 TO _NH_CFG DO
				IF aCfg[cf].rec > 0 THEN
					IF yFrm_235.DevToCat[cf] <> yFrm_235.DevToCat[0] THEN  				// oznacit, ci DEV vstupuje do nejakej CAT
						FOR i := 1 TO _Nh_CAT DO
							IF yFrm_235.DevToCat[cf].n[i] THEN
		      	         xA^.cat.cat[i] := true;                                         // SEC
							END_IF;

                  END_FOR;
					END_IF;
				END_IF;
         END_FOR;
		END_IF;
   	_Nh_FRM_Read(frm:=232);
		IF xA^.CatOk = false THEN
			// oznaci CAT, ktore maju nejake DEV
			FOR cf := 1 TO _Nh_CAT DO
				IF xA^.cat.cat[cf] THEN
					IF yFrm_232.CatToCat[cf] <> yFrm_232.CatToCat[0] THEN  				// DEV sa porovna s Empty, ma jejaku CAT
						FOR i := 1 TO _Nh_CAT DO
							IF yFrm_232.CatToCat[cf].n[i] THEN
      						xA^.cat.cat[i] := true;                                         // SEC
							END_IF;
						END_FOR;
            	END_IF;
				END_IF;
			END_FOR;
		END_IF;

//      xA^.cat.cat[35] := true;

		FOR nd := 1 TO USINT_TO_INT(_Nh_CAT) DO
			yes := yFrm_232.cat[nd].txt > 0;
			IF yes = false THEN
			ELSIF	xF^.typ  < 0 THEN
				yes := yFrm_232.CatToCat[xF^.typ].n[nd] AND (xA^.cat.cat[nd] OR xF^.typ =-2) ;  // podkategorie, ktore maju nejaky DEV alebo cely setup
			ELSIF xA^.cat.cat[nd] = false THEN
				yes := false;
			ELSIF xF^.cf.n > 0 THEN
				yes := yFrm_232.CatToCat[nd].n[xF^.cf.n];
			ELSE
				yes := false;
			END_IF;
			IF yes THEN
				CASE yFrm_232.cat[nd].rght OF                                // kto moze vidiet
    				1 :	yes := yes AND xA^.UsrRight > 0;
   	   	   2 :	yes := yes AND xA^.UsrRight > 1;
   	   	   3 :	yes := yes AND xA^.UsrRight > 2;
   	   	   9 :	yes := yes AND xA^.admin;
				END_CASE;

(*
				CASE yFrm_232.cat[nd].rght OF                                // kto moze vidiet
    				1 :	yes := yes AND xM^.set;
   	   	   2 :	yes := yes AND xA^.admin;
				END_CASE;
*)
				IF yes THEN
  					yIdxR          := _e_NH_IDX_ROW;
	   	      yIdxR.dev.c    := 2;
   	   	   yIdxR.dev.n    := nd;                                                // defaul sa pozije cislo vety
//   	      	yIdxR.dev.n    := 1;                                                // defaul sa pozije cislo vety
		   	   _NhCrIx(ok := yes);
				END_IF;
			END_IF;

	  	END_FOR;
	END_IF;

	IF xF^.dev.n[2] THEN																				// aj CAT do browsu
     	yIdxR          := _e_NH_IDX_ROW;
		yIdxR.dev.c    := 2;
		FOR i := 1 TO _Nh_CAT DO
			IF (xF^.cat.n[0] OR xF^.cat.n[i]) THEN //AND  xA^.cat.cat[i] THEN
            yIdxR.dev.n    := USINT_TO_INT(i);
			  _NhCrIx(ok := true);
			END_IF;
     	END_FOR;
	END_IF;

   IF xL^.vaz > 1 THEN                                                           // vazby, list
      _NhxPt(c := xF^.cf.c, n := xF^.cf.n,x:=35);
      xDev2          := xPt;
      // pri vstupe do browsu vazieb/lst resetne priznak pre dev v hlavicke. Vazby ich v dalsom cykle vratia spat ak tam budu
      nd             := 1;
      WHILE nd  <= aVaz[xL^.vaz].Rec DO                                         // vsetky vety CFG
         yIdxR          := _e_NH_IDX_ROW;
         IF _NhxVaz(cv := xL^.vaz, nd := nd ) THEN
            yIdxR          := _e_NH_IDX_ROW;
            yIdxR.chk      := 1;
            yIdxR.nd       := nd;
           	yIdxR.in  		:= 0;
           	yIdxR.vaz  		:= 1;
			   yes            := true;
																									// SCN=3 ACT=4
            IF xVaz^.in.c = xF^.cf.c AND xVaz^.in.n = xF^.cf.n THEN     	// hlavicka IN => riadok je OUT
	            yIdxR.dev := xVaz^.ou;
	           	yIdxR.in  := 0;
		      ELSIF xVaz^.OU.c = xF^.cf.c AND xVaz^.OU.n = xF^.cf.n THEN     // hlavicka OU => riadok je IN
            	yIdxR.in  := 1;
	            yIdxR.dev := xVaz^.IN;
				ELSE
					Yes := false;
				END_IF;
(*
				CASE xL^.vaz OF
      			3:	// SCN-list
		           	yIdxR.in  		:= false;
		            yIdxR.dev 		:= xVaz^.ou;
//	   	   		xDev2^.al.lst  := 1;
						aVaz[3].ref		:= true;
//        			4: // vazby TER,TEH,LUX... -> ROM
//   	   			xDev2^.al.lst  := 1;

        			4: // vazby ACT,ALA,BLK
		           	yIdxR.in  		:= false;
		            yIdxR.dev 		:= xVaz^.ou;
//   	   			xDev2^.al.lst  := 1;

(*
      		ELSE // 2 = WSB -> DEV
						IF yes THEN
							xDev2^.al.vaz  := 1;
						END_IF;
)
				END_CASE;
*)
				yes	:= yes AND xF^.dev.n[yIdxR.dev.c];

            IF xL^.fDv > 0 THEN
//               yes := yes AND xF^.dev.n[ yIdxR.dev.c ] ;                           // zapnuty fil=ter DEV
            END_IF;
            IF yes = false THEN
					;
				ELSIF xF^.rom > 0 THEN
               _NhxPt(c := yIdxR.dev.c, n := yIdxR.dev.n,x:=36);
               yes := xPt^.cf.rom = xF^.rom;                          // riadok ma ten isty rom ako hlavicka
            END_IF;
            IF yes THEN
               xPtU  := xIdx;                                           // zapamata si aktualny index
               xIdx  := xIdx1;                                          // nastavi sa na prvy index
               // hlada sa v indexe
               FOR i := 1 TO xIxB^.idx DO
                  IF xIdx^.ix[aWeb.nbr].dev.c = yIdxR.dev.c AND
                     xIdx^.ix[aWeb.nbr].dev.n = yIdxR.dev.n THEN
                     IF xIdx^.ix[aWeb.nbr].nd = 0 OR                    // tato veta nie je z vaz
                        xIdx^.ix[aWeb.nbr].nd = yIdxR.nd THEN           // je to tato ista veta
                        yes := false;
                        xIdx^.ix[aWeb.nbr].chk  := true;
                        xIdx^.ix[aWeb.nbr].vaz  := true;
                        xIdx^.ix[aWeb.nbr].in   := yIdxR.in;
                        xIdx^.ix[aWeb.nbr].nd   := yIdxR.nd;
                        EXIT;
                     END_IF;
                  END_IF;
                  xIdx := xIdx + SIZEOF(NH_IDX);
               END_FOR;
               xIdx := xPtU;                                            // vrati adresu aktualneho indexu
            END_IF;
            _NhCrIx(ok := yes);
         END_IF;
         nd := nd + 1;
      END_WHILE;
   END_IF;

   aSys.vIx2   := MAX(aSys.vIx2, aSys.vIx1 +  USINT_TO_UDINT(xIxB^.ofs) + USINT_TO_UDINT(xIxB^.idx) * SIZEOF(NH_IDX)); // najdlhsi koniec indexu
   IF aSys.vIx2 > _NH_RAM THEN // 65535 THEN
      aSys.Err_vIx2   := aSys.vIx2 - _NH_RAM;
   END_IF;

   _Nh_Brw_Idx   := xIxB^.idx > 0;                                                   // nieco nacitalo
   // vytvorit navigacne menu stranok
   IF xIxB^.idx > 0 THEN
      vr  		:= USINT_TO_REAL(xIxB^.idx) / USINT_TO_REAL(xIxB^.row.rws);				// zostane realne cislo s desatinou
		xIxB^.n	:= REAL_TO_USINT( CEIL(vr) );                                        // zaokruhli hore
      IF xIxB^.n > 1 THEN                                                           // bude vykreslovat gulicky stran
         xIxB^.w  := 40;
         xIxB^.x1 := (x2 - USINT_TO_INT(xIxB^.n-1) * 40)/2;
      ELSIF xIxB^.n > 0 THEN                                                              // bude vykreslovat gulicky stran
         xIxB^.x1 := x2/2;
      END_IF;
   END_IF;

(*
   IF xIxB^.idx > 0 THEN
      xIxB^.n  := USINT_TO_REAL(xIxB^.idx) / USINT_TO_REAL(xIxB^.row.rws);
      IF mod(xIxB^.idx,xIxB^.row.rws) > 0 THEN
         xIxB^.n  := xIxB^.n + 1;
      END_IF;
      IF xIxB^.n > 1 THEN                                                              // bude vykreslovat gulicky stran
         xIxB^.w  := 40;
         xIxB^.x1 := (x2 - USINT_TO_INT(xIxB^.n-1) * 40)/2;
      ELSIF xIxB^.n > 0 THEN                                                              // bude vykreslovat gulicky stran
         xIxB^.x1 := x2/2;
      END_IF;
   END_IF;
*)
   RETURN;
END_FUNCTION

FUNCTION _Nh_Frm_HOM {HIDDEN} : BOOL     // HOME menu
   VAR_TEMP
      brw      : bool;
      row      : USINT;
      obj      :  SINT;
      wht      :  SINT;
   END_VAR
   _Nh_Frm_HOM   := true;

//   xA^.usr     := 1;

//   _NhxUsr(u := xA^.usr);                                                 // namapuje usra

   CASE xM^.wht OF
     -1: ;

      1: // 1.kolo dolu (spat) = prekreslenie suradnic (animacia)
         xR := ADR(xB^.r[1]);
         FOR i := 1 TO 8 DO
            xR^.o.ob[i].x := _ePg0.xy[i].x;
            xR^.o.ob[i].y := REAL_TO_INT(INT_TO_REAL(_ePg0.xy[i].y)*yk);
         END_FOR;
         xA^.tch.cmd := 255;
         xM^.delay   := 50;
         xM^.wht     := -10;
         _Nh_Frm_HOM   := false;

      2: // 1.kolo hore (dalej) = prekreslenie suradnic (animacia)
         xR := ADR(xB^.r[1]);
         i := 8;
         WHILE i > 1 DO
            xR^.o.ob[i].x := _ePg0.xy[i-1].x;
            xR^.o.ob[i].y := REAL_TO_INT(INT_TO_REAL(_ePg0.xy[i-1].y)*yk);   //_ePg0.xy[i-1].y;
            i := i - 1;
         END_WHILE;
         xR^.o.ob[i].x := _ePg0.xy[8].x;
         xR^.o.ob[i].y := REAL_TO_INT(INT_TO_REAL(_ePg0.xy[8].y)*yk);   //_ePg0.xy[8].y;

         xA^.tch.cmd := 255;
         xM^.delay   := 50;
         xM^.wht     := -20;
         _Nh_Frm_HOM   := false;

     -10: // v 2.kole dolu
         IF _NhSet1Row(fnd := false, dn := true, row := xM^.ixb[0].row.rws ) THEN
            xUsr^.cx.ds1 := xL^.rw1;
         END_IF;
         brw := true;
//         wht := 25;

    -20: // v 2.kole hore
         IF _NhSet1Row(fnd := false, up := true, row := xM^.ixb[0].row.rws ) THEN
            xUsr^.cx.ds1 := xL^.rw1;
         END_IF;
         brw := true;
//         wht := 25;

      3: // dolava

      4: // doprava

     25: // nova stranka
         wht := 25;
//            _NhHomDat();

   END_CASE;

   CASE wht OF
      25:   // nacitat
//            _NhUsrPar(fav := 1, sav := 1, usr:=1 );
            xA^.fav  := xUsr^.cx.dsh;
            _Nh_Brw_Idx();
            xA^.fav  := xUsr^.cx.qck;
            _Nh_Brw_Idx(ixb := 1);
            xA^.fav  := xUsr^.cx.fav;
            brw      := true;

      1 : // dalej DASH
      2 : // spat DASH
      3 : // dalej QUICK
      4 : // spat QUICK
   ELSE     //xA^.fav := xUsr^.cx.qck;
            // _NhHomDat();
   END_CASE;

   IF brw THEN                                                    // naplni browser podla 1.row
(*
      NH_EMPTY : NH_HOM_DSH ;             // 0    rezeva
      DSH      : NH_HOM_DSH ;             // 1     DASH
      QCK      : NH_HOM_QCK ;             // 2     Quick-menu
      HOM      : NH_HOM_HOM ;             // 3     domcek s okolim
      LUP      : NH_HOM_LUP ;             // 4     objekt k DSH vlavo hore
      PUP      : NH_HOM_PUP ;             // 5     objekt k DSH vpravo hore
      LDN      : NH_HOM_LDN ;             // 6     objekt k DSH vlavo dolu
      PDN      : NH_HOM_PDN ;             // 7     objekt k DSH vpravo dolu
      WHT      : NH_HOM_WHT ;             // 8     wheater
      OTH      : NH_HOM_OTH ;             // 9     ostatne

*)
      _NheBrw( wht := 5);                                         		// vymaze data LEN brw
      _Nh_FRM_Read(frm:=11);
      xPtD  := ADR(xB^.r[9].o.ob[1].cf.n); 	      // adresa premennej USINT;
      xPtD^ := PTR_TO_UDINT(ADR(xHom^.cx.pDay));	      // adresa xPod aktualneho domceka/bytu

      IF yk > 1.0 THEN
         FOR i := 1 TO 7 DO
            xR    := ADR(xB^.r[ i ]);
            FOR jj := 0 TO _RowObr DO
               IF i=2 THEN
                  ix :=100;
               ELSE
                  ix := 70;
               END_IF;
               xR^.o.ob[jj].y := xR^.o.ob[jj].y + ix; //REAL_TO_INT( INT_TO_REAL(xR^.o.ob[jj].y) * yk );
            END_FOR;
         END_FOR;
      END_IF;
      FOR j := 0 TO 1 DO
         IF _Nh_Map_Idx(ixb := SINT_TO_USINT(j)) THEN
            ii := MIN(xIxB^.idx,xIxB^.row.rws);
            IF j = 0 THEN                                            // DASH
               xR := ADR(xB^.r[ 1 ]);
               xL^.rw1  := xUsr^.cx.ds1;                             // nacita poslene zapamatany 1.DEV pre aktualneho usra
               IF _NhSet1Row(ixb := 0 ) THEN
                  xUsr^.cx.ds1 := xL^.rw1;                           // zapamata si novy, alebo povodny DEV
               END_IF;
            ELSE                                                     // QUICK
               xR := ADR(xB^.r[ 2 ]);
               xL^.rw1  := xUsr^.cx.qc1;                             // nacita poslene zapamatany 1.DEV pre aktualneho usra
               IF _NhSet1Row(ixb := 1 ) THEN
                  xUsr^.cx.qc1 := xL^.rw1;                           // zapamata si novy, alebo povodny DEV
               END_IF;
            END_IF;
            xIxB^.ix1 := 1;
            xIxB^.ix2 := 0;
            FOR i := 1 TO ii DO
               xR^.o.ob[i].cf := xIdx^.ix[aWeb.nbr].dev;
               cf := xR^.o.ob[i].cf.c;
               IF cf =  2 THEN                  xR^.o.ob[i].wh := 232;     // obrazok z CAT-stat
               ELSE                             xR^.o.ob[i].wh := 233;     // obrazok z DEV / sekcie QCK
               END_IF;
               xIxB^.ix2      := xIxB^.ix2 + 1;
               xIdx           := xIdx + SIZEOF(NH_IDX);
            END_FOR;
         ELSE
            xIxB^.ix1 := 0;
            xIxB^.ix2 := 0;
         END_IF;
      END_FOR;
      xL^.rw1  := xUsr^.cx.ds1;                             // zapamatany DEV v 1.riadku pre usra
   END_IF;

   GC_Begin(GrData := xCan);
//   aSys.cnt    := aSys.cnt + 1;
   row := 1;
   WHILE row <= _RowBrw DO
      xR := ADR(xB^.r[ row  ]);
      IF true THEN //xR^.h.nd > 0 THEN
         obj := 0;
         WHILE obj <= _RowObr DO
            IF xR^.o.ob[obj].wh > 0 THEN
               IF xL^.obj = 0 THEN										// home page
                 	_NhxCfg(c := xF^.cf.c, n := xF^.cf.n, x:=43);                     // xDev,xCfg,xPar pre aktualny riadok
					ELSIF xR^.o.ob[obj].cf.c = 2 OR xR^.o.ob[obj].wh = 107 THEN
						;
               ELSIF xR^.o.ob[obj].cf.c > 0 AND xR^.o.ob[obj].cf.n > 0 THEN
                  _NhxCfg(c := xR^.o.ob[obj].cf.c, n := xR^.o.ob[obj].cf.n,x:=43);                     // xDev,xCfg,xPar pre aktualny riadok
               ELSIF row = 1 THEN
						;
               END_IF;
               _Nh_Shw_Obj(row:=row, obj := obj);                       // zobrazi 1.objekt a necha namapovane xO
            END_IF;
            obj := obj + 1;
         END_WHILE;
      END_IF;
      row := row + 1;
   END_WHILE;

   _NhShwMnu();
   GC_End(GrData := xCan);

END_FUNCTION

{ $ END_IF }
